(* CODESYS project kod + gui.project
   Title: seminarski
   Version: 0.0.0.0
   Author: Kemal

Project tree, tasks and I/O mapping:
  MyController : TM238LDD24DT, Schneider Electric, order no. TM238LDD24DT, version 4.0.1.28
      settings: OpcUa Enable = False
    application Application
      task MAST (cyclic, interval 20 ms, priority 15, watchdog 100 ms x 1) calls main, testiranje, izmjene, razlike
      global variables GVL
      program testiranje [ST]
      program main [ST]
      Symbols
      program izmjene [ST]
      program razlike [ST]
    Embedded Functions
      IO : IO, Schneider Electric, version 4.0.1.28
          input  Application.I_start : BOOL  // IW0.I0
          input  Application.I_stop : BOOL  // IW0.I1
          input  Application.Q[counter,3] : BOOL  // IW0.I3
          input  Application.Q[counter,4] : BOOL  // IW0.I4
          input  Application.Q[counter,5] : BOOL  // IW0.I5
          input  Application.Q[counter,6] : BOOL  // IW0.I6
          input  Application.Q[counter,7] : BOOL  // IW0.I7
          output Application.Q_0 : BOOL  // QW0.Q0
          output Application.Q_1 : BOOL  // QW0.Q1
          output Application.Q_2 : BOOL  // QW0.Q2
          output Application.Q_red_LED : BOOL  // QW0.Q4
          output Application.Q_yellow_LED : BOOL  // QW0.Q5
          output Application.Q_green_LED : BOOL  // QW0.Q6
          unmapped channels: IW0, QW0
      HSC : HSC, Schneider Electric, version 4.0.1.28
      PTO_PWM : PTO_PWM, Schneider Electric, version 4.0.1.28
    Serial Line
      SoMachine_Network_Manager : SoMachine-Network Manager, Schneider Electric, version 4.0.0.2
  HMIS5T : HMIS5T, Schneider Electric, order no. HMIS5T, version 3.5.3.54
    HMI Application
    COM1
      SoMachine_Network_Manager1 : SoMachine-Network Manager, Schneider Electric, version 4.0.0.2
    Ethernet
      SoMachine_Network_Manager2 : SoMachine-Network Manager, Schneider Electric, version 4.0.0.2
    USB
      SoMachine_Network_Manager3 : SoMachine-Network Manager, Schneider Electric, version 4.0.0.2
  Vijeo Designer Project Container Data
  Vijeo Designer Project Container
*)

// MyController/Application/GVL
VAR_GLOBAL
END_VAR
VAR_GLOBAL
	main_menu: BOOL;
	signals_menu: BOOL;
	timers_menu: BOOL;
	test: BOOL;
	stop: BOOL;
	counter: INT := -42;
	I_start: BOOL;
	I_stop: BOOL;
	Q_0: BOOL;
	Q_1: BOOL;
	Q_2: BOOL;
	I_3: BOOL;
	I_4: BOOL;
	I_5: BOOL;
	I_6: BOOL;
	I_7: BOOL;
	Q: ARRAY[0..7, 3..7] OF BOOL := [TRUE, 2(FALSE), TRUE, 2(FALSE), TRUE, FALSE, TRUE, 3(FALSE), 2(TRUE), FALSE, TRUE, 3(FALSE), TRUE, FALSE, TRUE, 2(FALSE), TRUE, 2(FALSE), TRUE, FALSE, TRUE, 3(FALSE), 4(TRUE), FALSE, 2(TRUE)];
	Q_red_LED: BOOL;
	Q_yellow_LED: BOOL;
	Q_green_LED: BOOL;
END_VAR

// MyController/Application/main
PROGRAM main
VAR
	timer: TP;
	ukini_red_LED: BOOL;
	vakat: REAL := 3;
END_VAR

Q_yellow_LED := test;

timer(IN := stop, PT := REAL_TO_TIME(1000*vakat));
IF timer.Q THEN
	RETURN;
END_IF
stop := FALSE;
IF ukini_red_LED THEN
	Q_red_LED := FALSE;
	counter := -42;
	ukini_red_LED := FALSE;
END_IF

main_menu := NOT (signals_menu OR timers_menu OR test OR stop OR Q_red_LED OR Q_green_LED);

IF I_start AND main_menu THEN
	counter := 0;
	Q_0 := counter.0;
	Q_1 := counter.1;
	Q_2 := counter.2;
	I_3 := Q[counter,3];
	I_4 := Q[counter,4];
	I_5 := Q[counter,5];
	I_6 := Q[counter,6];
	I_7 := Q[counter,7];
	test := TRUE;
END_IF

IF I_stop AND test THEN
	test := FALSE;
	stop := TRUE;
	ukini_red_LED := TRUE;
END_IF

END_PROGRAM

// MyController/Application/testiranje
PROGRAM testiranje
VAR
	timer: TON;
	vakat: REAL := 1;
END_VAR

timer(IN := test, PT := REAL_TO_TIME(1000*vakat));
IF NOT timer.Q THEN
	RETURN;
END_IF
timer(IN := FALSE);

IF I_3 <> Q[counter,3] OR I_4 <> Q[counter,4] OR I_5 <> Q[counter,5] OR I_6 <> Q[counter,6] OR I_7 <> Q[counter,7] THEN
	Q_red_LED := TRUE;
END_IF

counter := counter + 1;

Q_0 := counter.0;
Q_1 := counter.1;
Q_2 := counter.2;

IF counter = 8 THEN
	counter := 42;
	test := FALSE;
	IF NOT Q_red_LED THEN
		Q_green_LED := TRUE;
	END_IF
	RETURN;
END_IF

I_3 := Q[counter,3];
I_4 := Q[counter,4];
IF counter = 3 THEN
	I_4 := TRUE;
END_IF
I_5 := Q[counter,5];
I_6 := Q[counter,6];
IF counter = 6 THEN
	I_6 := FALSE;
END_IF
I_7 := Q[counter,7];

END_PROGRAM

// MyController/Application/izmjene
PROGRAM izmjene
VAR
	Q03: BOOL := Q[0,3];
	Q04: BOOL := Q[0,4];
	Q05: BOOL := Q[0,5];
	Q06: BOOL := Q[0,6];
	Q07: BOOL := Q[0,7];
	Q13: BOOL := Q[1,3];
	Q14: BOOL := Q[1,4];
	Q15: BOOL := Q[1,5];
	Q16: BOOL := Q[1,6];
	Q17: BOOL := Q[1,7];
	Q23: BOOL := Q[2,3];
	Q24: BOOL := Q[2,4];
	Q25: BOOL := Q[2,5];
	Q26: BOOL := Q[2,6];
	Q27: BOOL := Q[2,7];
	Q33: BOOL := Q[3,3];
	Q34: BOOL := Q[3,4];
	Q35: BOOL := Q[3,5];
	Q36: BOOL := Q[3,6];
	Q37: BOOL := Q[3,7];
	Q43: BOOL := Q[4,3];
	Q44: BOOL := Q[4,4];
	Q45: BOOL := Q[4,5];
	Q46: BOOL := Q[4,6];
	Q47: BOOL := Q[4,7];
	Q53: BOOL := Q[5,3];
	Q54: BOOL := Q[5,4];
	Q55: BOOL := Q[5,5];
	Q56: BOOL := Q[5,6];
	Q57: BOOL := Q[5,7];
	Q63: BOOL := Q[6,3];
	Q64: BOOL := Q[6,4];
	Q65: BOOL := Q[6,5];
	Q66: BOOL := Q[6,6];
	Q67: BOOL := Q[6,7];
	Q73: BOOL := Q[7,3];
	Q74: BOOL := Q[7,4];
	Q75: BOOL := Q[7,5];
	Q76: BOOL := Q[7,6];
	Q77: BOOL := Q[7,7];
END_VAR

Q[0,3] := Q03;
Q[0,4] := Q04;
Q[0,5] := Q05;
Q[0,6] := Q06;
Q[0,7] := Q07;
Q[1,3] := Q13;
Q[1,4] := Q14;
Q[1,5] := Q15;
Q[1,6] := Q16;
Q[1,7] := Q17;
Q[2,3] := Q23;
Q[2,4] := Q24;
Q[2,5] := Q25;
Q[2,6] := Q26;
Q[2,7] := Q27;
Q[3,3] := Q33;
Q[3,4] := Q34;
Q[3,5] := Q35;
Q[3,6] := Q36;
Q[3,7] := Q37;
Q[4,3] := Q43;
Q[4,4] := Q44;
Q[4,5] := Q45;
Q[4,6] := Q46;
Q[4,7] := Q47;
Q[5,3] := Q53;
Q[5,4] := Q54;
Q[5,5] := Q55;
Q[5,6] := Q56;
Q[5,7] := Q57;
Q[6,3] := Q63;
Q[6,4] := Q64;
Q[6,5] := Q65;
Q[6,6] := Q66;
Q[6,7] := Q67;
Q[7,3] := Q73;
Q[7,4] := Q74;
Q[7,5] := Q75;
Q[7,6] := Q76;
Q[7,7] := Q77;

END_PROGRAM

// MyController/Application/razlike
PROGRAM razlike
VAR
	timer: TP;
	vakat: REAL := 7;
	Q03: BOOL;
	Q04: BOOL;
	Q05: BOOL;
	Q06: BOOL;
	Q07: BOOL;
	Q13: BOOL;
	Q14: BOOL;
	Q15: BOOL;
	Q16: BOOL;
	Q17: BOOL;
	Q23: BOOL;
	Q24: BOOL;
	Q25: BOOL;
	Q26: BOOL;
	Q27: BOOL;
	Q33: BOOL;
	Q34: BOOL;
	Q35: BOOL;
	Q36: BOOL;
	Q37: BOOL;
	Q43: BOOL;
	Q44: BOOL;
	Q45: BOOL;
	Q46: BOOL;
	Q47: BOOL;
	Q53: BOOL;
	Q54: BOOL;
	Q55: BOOL;
	Q56: BOOL;
	Q57: BOOL;
	Q63: BOOL;
	Q64: BOOL;
	Q65: BOOL;
	Q66: BOOL;
	Q67: BOOL;
	Q73: BOOL;
	Q74: BOOL;
	Q75: BOOL;
	Q76: BOOL;
	Q77: BOOL;
	podudarnost_Q0: BOOL;
	podudarnost_Q1: BOOL;
	podudarnost_Q2: BOOL;
	podudarnost_Q3: BOOL;
	podudarnost_Q4: BOOL;
	podudarnost_Q5: BOOL;
	podudarnost_Q6: BOOL;
	podudarnost_Q7: BOOL;
END_VAR

CASE counter OF
0 : Q03 := I_3 XOR Q[0,3];
	Q04 := I_4 XOR Q[0,4];
	Q05 := I_5 XOR Q[0,5];
	Q06 := I_6 XOR Q[0,6];
	Q07 := I_7 XOR Q[0,7];
	podudarnost_Q0 := NOT (Q03 OR Q04 OR Q05 OR Q06 OR Q07);
1 : Q13 := I_3 XOR Q[1,3];
	Q14 := I_4 XOR Q[1,4];
	Q15 := I_5 XOR Q[1,5];
	Q16 := I_6 XOR Q[1,6];
	Q17 := I_7 XOR Q[1,7];
	podudarnost_Q1 := NOT (Q13 OR Q14 OR Q15 OR Q16 OR Q17);
2 : Q23 := I_3 XOR Q[2,3];
	Q24 := I_4 XOR Q[2,4];
	Q25 := I_5 XOR Q[2,5];
	Q26 := I_6 XOR Q[2,6];
	Q27 := I_7 XOR Q[2,7];
	podudarnost_Q2 := NOT (Q23 OR Q24 OR Q25 OR Q26 OR Q27);
3 : Q33 := I_3 XOR Q[3,3];
	Q34 := I_4 XOR Q[3,4];
	Q35 := I_5 XOR Q[3,5];
	Q36 := I_6 XOR Q[3,6];
	Q37 := I_7 XOR Q[3,7];
	podudarnost_Q3 := NOT (Q33 OR Q34 OR Q35 OR Q36 OR Q37);
4 : Q43 := I_3 XOR Q[4,3];
	Q44 := I_4 XOR Q[4,4];
	Q45 := I_5 XOR Q[4,5];
	Q46 := I_6 XOR Q[4,6];
	Q47 := I_7 XOR Q[4,7];
	podudarnost_Q4 := NOT (Q43 OR Q44 OR Q45 OR Q46 OR Q47);
5 : Q53 := I_3 XOR Q[5,3];
	Q54 := I_4 XOR Q[5,4];
	Q55 := I_5 XOR Q[5,5];
	Q56 := I_6 XOR Q[5,6];
	Q57 := I_7 XOR Q[5,7];
	podudarnost_Q5 := NOT (Q53 OR Q54 OR Q55 OR Q56 OR Q57);
6 : Q63 := I_3 XOR Q[6,3];
	Q64 := I_4 XOR Q[6,4];
	Q65 := I_5 XOR Q[6,5];
	Q66 := I_6 XOR Q[6,6];
	Q67 := I_7 XOR Q[6,7];
	podudarnost_Q6 := NOT (Q63 OR Q64 OR Q65 OR Q66 OR Q67);
7 : Q73 := I_3 XOR Q[7,3];
	Q74 := I_4 XOR Q[7,4];
	Q75 := I_5 XOR Q[7,5];
	Q76 := I_6 XOR Q[7,6];
	Q77 := I_7 XOR Q[7,7];
	podudarnost_Q7 := NOT (Q73 OR Q74 OR Q75 OR Q76 OR Q77);
42: IF Q_red_LED THEN
		timer(IN := TRUE, PT := REAL_TO_TIME(1000*vakat));
	ELSE
		timer(IN := TRUE, PT := REAL_TO_TIME(1000*vakat*3/5));
	END_IF
	IF timer.Q THEN
		RETURN;
	END_IF
	timer(IN := FALSE);
	Q_red_LED := FALSE;
	Q_green_LED := FALSE;
	counter := -42;
END_CASE

END_PROGRAM
